// TwinCAT 3 PLC project Array_Reset
// ProgramVersion: 3.1.4026.16
// libraries:
//   Tc2_Standard, * (Beckhoff Automation GmbH)
//   Tc2_System, * (Beckhoff Automation GmbH)
// project tree:
//   / PlcTask.TcTTO
//   POUs/ FB_DataSim.TcPOU, FB_Messwerte.TcPOU, FC_ResetArray.TcPOU, MAIN.TcPOU
// (motion and I/O tree: see PLC project hausaufgaben_flipflop)
// real-time tasks:
//   TASK PlcTask: cycle T#10ms, priority 20, ADS port 350
//   TASK PlcTask1: cycle T#10ms, priority 21, ADS port 351
//   TASK PlcTask2: cycle T#10ms, priority 22, ADS port 352
//   TASK PlcTask3: cycle T#10ms, priority 23, ADS port 353

CONFIGURATION Array_Reset
    RESOURCE PLC ON TwinCAT3
        TASK PlcTask(INTERVAL := T#10ms, PRIORITY := 23);
        PROGRAM MAIN WITH PlcTask : MAIN;
    END_RESOURCE
END_CONFIGURATION

// ---- POUs/MAIN.TcPOU
PROGRAM MAIN
VAR
	DataSim: FB_DataSim;
END_VAR

DataSim();

END_PROGRAM

// ---- POUs/FB_DataSim.TcPOU
FUNCTION_BLOCK FB_DataSim
VAR_INPUT
END_VAR
VAR_OUTPUT
	rValue: REAL := 1.0000;
END_VAR
VAR
	CountTimer: TON;
	RisingEdge: R_TRIG;
	DataStack: FB_Messwerte;
END_VAR

CountTimer(IN := TRUE, PT := T#2S);
RisingEdge(CLK:= CountTimer.Q);

IF RisingEdge.Q AND rValue < 10000 THEN
	rValue := rValue * LREAL_TO_REAL(PI);
	DataStack(rValue := rValue);
ELSIF RisingEdge.Q AND rValue > 10000 THEN
	rValue := (rValue /100) * 1.75;
	DataStack(rValue := rValue);
END_IF

IF CountTimer.Q THEN
	CountTimer(IN := FALSE);
	CountTimer(IN := TRUE);
END_IF

END_FUNCTION_BLOCK

// ---- POUs/FB_Messwerte.TcPOU
FUNCTION_BLOCK FB_Messwerte
VAR_INPUT
	Ix_Reset: BOOL;
	rValue: REAL;
END_VAR
VAR_OUTPUT
END_VAR
VAR
	Messwerte: ARRAY[1..20] OF REAL;
	iInPos: INT:= 1;
	vsx_FP_Reset: BOOL;
END_VAR

IF Ix_Reset AND NOT vsx_FP_Reset THEN
FC_ResetArray(Ix_Reset:= Ix_Reset, Messwerte := Messwerte);
END_IF

Messwerte[iInPos] := rValue;

IF iInPos >= 20 THEN
	iInPos := 1;
ELSE
	iInpos := iInPos +1;
END_IF

vsx_FP_Reset := Ix_Reset;

END_FUNCTION_BLOCK

// ---- POUs/FC_ResetArray.TcPOU
FUNCTION FC_ResetArray : BOOL
VAR_INPUT
	Ix_Reset: BOOL;
END_VAR
VAR_STAT
	vsx_FP_Reset: BOOL;
END_VAR
VAR
	vti_Index: INT := 1;
	iCounter: INT := 1;
END_VAR
VAR_IN_OUT
	Messwerte: Array[1..20] OF REAL;
END_VAR

	FOR iCounter := 1 TO 20 DO
		Messwerte[vti_Index] := 0;
	END_FOR

END_FUNCTION
